FUNCTION_BLOCK EM_Machine IMPLEMENTS  ITF_PackMLV2
VAR_INPUT
END_VAR
VAR_OUTPUT
END_VAR
VAR
	fb_mem	: STRUCT_EM_Machine;
	ton1	: ton;
END_VAR

(*
$$$$$$$$\                                                                   $$\       $$$$$$$$\                     $$\                                         $$\                     
$$  _____|                                                                  $$ |      $$  _____|                    \__|                                        \__|                    
$$ |   $$$$$$\   $$$$$$\  $$$$$$$\  $$\  $$\  $$\  $$$$$$\   $$$$$$\   $$$$$$$ |      $$ |      $$$$$$$\   $$$$$$\  $$\ $$$$$$$\   $$$$$$\   $$$$$$\   $$$$$$\  $$\ $$$$$$$\   $$$$$$\  
$$$$$\ \____$$\ $$  __$$\ $$  __$$\ $$ | $$ | $$ |$$  __$$\ $$  __$$\ $$  __$$ |      $$$$$\    $$  __$$\ $$  __$$\ $$ |$$  __$$\ $$  __$$\ $$  __$$\ $$  __$$\ $$ |$$  __$$\ $$  __$$\ 
$$  __|$$$$$$$ |$$ |  \__|$$ |  $$ |$$ | $$ | $$ |$$ /  $$ |$$ /  $$ |$$ /  $$ |      $$  __|   $$ |  $$ |$$ /  $$ |$$ |$$ |  $$ |$$$$$$$$ |$$$$$$$$ |$$ |  \__|$$ |$$ |  $$ |$$ /  $$ |
$$ |  $$  __$$ |$$ |      $$ |  $$ |$$ | $$ | $$ |$$ |  $$ |$$ |  $$ |$$ |  $$ |      $$ |      $$ |  $$ |$$ |  $$ |$$ |$$ |  $$ |$$   ____|$$   ____|$$ |      $$ |$$ |  $$ |$$ |  $$ |
$$ |  \$$$$$$$ |$$ |      $$ |  $$ |\$$$$$\$$$$  |\$$$$$$  |\$$$$$$  |\$$$$$$$ |      $$$$$$$$\ $$ |  $$ |\$$$$$$$ |$$ |$$ |  $$ |\$$$$$$$\ \$$$$$$$\ $$ |      $$ |$$ |  $$ |\$$$$$$$ |
\__|   \_______|\__|      \__|  \__| \_____\____/  \______/  \______/  \_______|      \________|\__|  \__| \____$$ |\__|\__|  \__| \_______| \_______|\__|      \__|\__|  \__| \____$$ |
                                                                                                          $$\   $$ |                                                          $$\   $$ |
                                                                                                          \$$$$$$  |                                                          \$$$$$$  |
                                                                                                           \______/                                                            \______/ 
*)
//********************************Initiating***********************************
fb_mem.STS.State := PackML_StateMachine(State			:= fb_mem.STS.State,
										Start           := fb_mem.CS.Start,
										Stop            := fb_mem.CS.Stop,
										Reset           := fb_mem.CS.Reset,
										Abort           := fb_mem.CS.Abort,
										Clear           := fb_mem.CS.Clear,
										UnSuspend       := fb_mem.CS.UnSuspend,
										Suspend         := fb_mem.CS.Suspend,
										UnHold          := fb_mem.CS.UnHold,
										Hold            := fb_mem.CS.Hold,
										Starting_SC     := fb_mem.STS.Starting_SC,
										Execute_SC      := fb_mem.STS.Execute_SC,
										Completing_SC	:= fb_mem.STS.Completing_SC,
										Resetting_SC    := fb_mem.STS.Resetting_SC,
										Holding_SC      := fb_mem.STS.Holding_SC,
										Unholding_SC    := fb_mem.STS.Unholding_SC,
										Suspending_SC   := fb_mem.STS.Suspending_SC,
										Unsuspending_SC := fb_mem.STS.Unsuspending_SC,
										Aborting_SC     := fb_mem.STS.Aborting_SC,
										Clearing_SC     := fb_mem.STS.Clearing_SC,
										Stopping_SC     := fb_mem.STS.Stopping_SC);
										
//********************************ZEROING***********************************								
fb_mem.STS.Starting_SC 		:= FALSE;
fb_mem.STS.Execute_SC 		:= FALSE;
fb_mem.STS.Resetting_SC 	:= FALSE;
fb_mem.STS.Holding_SC 		:= FALSE;
fb_mem.STS.Unholding_SC 	:= FALSE;
fb_mem.STS.Suspending_SC 	:= FALSE;
fb_mem.STS.Unsuspending_SC 	:= FALSE;
fb_mem.STS.Aborting_SC 		:= FALSE;
fb_mem.STS.Clearing_SC 		:= FALSE;
fb_mem.STS.Stopping_SC 		:= FALSE;
fb_mem.STS.Completing_SC 	:= FALSE;

//********************************Auto manual logic***********************************
IF fb_mem.CS.Auto OR fb_mem.HMI.Auto THEN
	fb_mem.STS.Auto := TRUE;
	fb_mem.STS.Manueel := FALSE;
END_IF

IF fb_mem.CS.Manueel OR fb_mem.HMI.Manueel THEN
	fb_mem.STS.Auto := FALSE;
	fb_mem.STS.Manueel := TRUE;
END_IF

//********************************Action case***********************************

// THIS CODE SIMULATES A EXTERNAL MACHINE WICH RUNS ON PACKML. SO NO ACTION CASE IS PROGRAMMED


//********************************HMI_Connection***********************************
fb_mem.STS.StringState     := TO_STRING(fb_mem.STS.State); 

//********************************ZEROING***********************************

fb_mem.CS.Auto            := FALSE;
fb_mem.CS.Manueel         := FALSE;
fb_mem.CS.Start           := FALSE;
fb_mem.CS.Stop            := FALSE;
fb_mem.CS.Reset           := FALSE;
fb_mem.CS.Abort           := FALSE;
fb_mem.CS.Clear           := FALSE;
fb_mem.CS.UnSuspend       := FALSE;
fb_mem.CS.Suspend         := FALSE;
fb_mem.CS.UnHold          := FALSE;
fb_mem.CS.Hold            := FALSE;

{warning 'add method implementation '}
METHOD Abort : BOOL
fb_mem.CS.Abort := TRUE;
END_METHOD

METHOD Aborting_SC : BOOL
VAR_INPUT
END_VAR
fb_mem.STS.Aborting_SC := TRUE;
END_METHOD

{warning 'add method implementation '}
METHOD Auto : BOOL
fb_mem.CS.Auto := TRUE;
Auto := fb_mem.STS.Auto;
END_METHOD

{warning 'add method implementation '}
METHOD Clear : BOOL
fb_mem.CS.Clear := TRUE;
END_METHOD

METHOD Clearing_SC : BOOL
VAR_INPUT
END_VAR
fb_mem.STS.Clearing_SC := TRUE;
END_METHOD

METHOD Completing_SC : BOOL
VAR_INPUT
END_VAR
fb_mem.STS.Completing_SC := TRUE;
END_METHOD

METHOD Execute_SC : BOOL
VAR_INPUT
END_VAR
fb_mem.STS.Execute_SC := TRUE;
END_METHOD

METHOD FB_init : BOOL
VAR_INPUT
	bInitRetains : BOOL; // if TRUE, the retain variables are initialized (warm start / cold start)
	bInCopyCode : BOOL;  // if TRUE, the instance afterwards gets moved into the copy code (online change)
END_VAR
//**************************INITIATE**************************//
END_METHOD

{warning 'add method implementation '}
METHOD Hold : BOOL
fb_mem.CS.Hold := TRUE;
END_METHOD

METHOD Holding_SC : BOOL
VAR_INPUT
END_VAR
fb_mem.STS.Holding_SC := TRUE;
END_METHOD

{warning 'add method implementation '}
METHOD Manueel : BOOL
fb_mem.CS.Manueel := TRUE;
Manueel := fb_mem.STS.Manueel;
END_METHOD

{warning 'add method implementation '}
METHOD Reset : BOOL
fb_mem.CS.Reset := TRUE;
END_METHOD

METHOD Resetting_SC : BOOL
VAR_INPUT
END_VAR
fb_mem.STS.Resetting_SC := TRUE;
END_METHOD

{warning 'add method implementation '}
METHOD Start : BOOL
fb_mem.CS.Start := TRUE;
END_METHOD

METHOD Starting_SC : BOOL
VAR_INPUT
END_VAR
fb_mem.STS.Starting_SC := TRUE;
END_METHOD

{warning 'add property implementation'}
PROPERTY State : E_State_PackML
GET
State := fb_mem.STS.State;
END_GET
END_PROPERTY

{warning 'add method implementation '}
METHOD Stop : BOOL
fb_mem.CS.Stop := TRUE;
END_METHOD

METHOD Stopping_SC : BOOL
VAR_INPUT
END_VAR
fb_mem.STS.Stopping_SC := TRUE;
END_METHOD

{warning 'add method implementation '}
METHOD Suspend : BOOL
fb_mem.CS.Suspend := TRUE;
END_METHOD

METHOD Suspending_SC : BOOL
VAR_INPUT
END_VAR
fb_mem.STS.Suspending_SC := TRUE;
END_METHOD

{warning 'add method implementation '}
METHOD Unhold : BOOL
fb_mem.CS.Unhold := TRUE;
END_METHOD

METHOD Unholding_SC : BOOL
VAR_INPUT
END_VAR
fb_mem.STS.Unholding_SC := TRUE;
END_METHOD

{warning 'add method implementation '}
METHOD Unsuspend : BOOL
fb_mem.CS.Unsuspend := TRUE;
END_METHOD

METHOD Unsuspending_SC : BOOL
VAR_INPUT
END_VAR
fb_mem.STS.Unsuspending_SC := TRUE;
END_METHOD

{warning 'add method implementation '}
METHOD ZeroAllVar : BOOL
END_METHOD

END_FUNCTION_BLOCK

(* stored: Version 1.1.0.1, ProductVersion 3.1.4024.12
   POU EM_Machine: Id {0ded22b0-cd36-4d7d-bc24-4ace5391502f}, SpecialFunc None
   Folder Methods: Id {880b40f2-88eb-491a-87ab-b85a58b2e18b}
   Folder Properties: Id {00f11200-79c1-4854-9fd3-409f054934e7}
   Method Abort: Id {f5b473a4-f483-4f65-bb76-a50b980f4490}
   Method Aborting_SC: Id {2e1f91a2-c54e-4083-aad9-252cd9c83e70}
   Method Auto: Id {5f124478-c8ce-4452-a23b-4bbae3ba6710}
   Method Clear: Id {6b030e6b-ccce-4524-902a-2a45764d4629}
   Method Clearing_SC: Id {67748f50-5a3e-48c5-850b-a96247c04a26}
   Method Completing_SC: Id {f855bb44-5cdb-42d7-afe8-d162963806ab}
   Method Execute_SC: Id {78c3844e-5af5-4337-b93e-3d3a1da3e38c}
   Method FB_init: Id {232cf6e5-cfd3-4138-9681-ea49b1ba5424}
   Method Hold: Id {8470fcbb-be12-4179-8327-f37f71178635}
   Method Holding_SC: Id {2d03bc99-2f15-4fb7-a6a2-0ec9455ed642}
   Method Manueel: Id {239b93df-25e0-43af-a662-6a0df2b8c7cd}
   Method Reset: Id {d05bb64c-63e5-48c3-9a1e-d8d06d22b460}
   Method Resetting_SC: Id {c9f22d73-7395-4123-ad63-7b653740f97b}
   Method Start: Id {08ad76fe-a4a1-4453-9531-7b051762e226}
   Method Starting_SC: Id {cd518995-e0e9-4034-82df-a1c6d0dbd27c}
   Property State: Id {b7d438e7-0251-4721-9efc-d6f6cb6aa6ac}
   Get Get: Id {db4e1595-0897-4a61-b676-50ce21282e5b}
   Method Stop: Id {87e4bc3d-3ef7-42ec-8db5-7cd3e3b97d56}
   Method Stopping_SC: Id {888f0238-9b7d-4394-9cdb-3c4ae3070ccc}
   Method Suspend: Id {3703d8f0-d4e2-498b-9c83-7435fdeecfee}
   Method Suspending_SC: Id {cad620d4-5436-4978-aa63-b54fc64d6877}
   Method Unhold: Id {ba06b9f5-6ede-47b3-bdfa-a0ae6183e169}
   Method Unholding_SC: Id {333f9b51-82f7-4d93-b050-62fea770f886}
   Method Unsuspend: Id {850d5016-ac19-411e-a144-7720a100df80}
   Method Unsuspending_SC: Id {673da040-0d86-4561-846e-b7cdfb7fc49a}
   Method ZeroAllVar: Id {700871ed-e48a-4a68-834f-3719580aa532} *)
